// TwinCAT 3 PLC project PLC1
// ProgramVersion: 3.1.4024.0
// libraries:
//   Tc2_Standard, * (Beckhoff Automation GmbH)
//   Tc2_System, * (Beckhoff Automation GmbH)
//   Tc3_IotCommunicator, * (Beckhoff Automation GmbH)
//   Tc3_Module, * (Beckhoff Automation GmbH)
// project tree:
//   DUTs/ ST_Mqtt_Data.TcDUT
//   / PlcTask.TcTTO
//   POUs/ MAIN.TcPOU
// real-time tasks:
//   TASK PlcTask: cycle T#10ms, priority 20, ADS port 350

CONFIGURATION PLC1
    RESOURCE PLC ON TwinCAT3
        TASK PlcTask(INTERVAL := T#10ms, PRIORITY := 20);
        PROGRAM MAIN WITH PlcTask : MAIN;
    END_RESOURCE
END_CONFIGURATION

// ---- DUTs/ST_Mqtt_Data.TcDUT
TYPE ST_Mqtt_Data :
STRUCT
	{attribute 'iot.DisplayName' := 'Valve'}
	valve1 : BOOL;
	{attribute 'iot.DisplayName' := 'Pressure Transducer'}
    {attribute 'iot.ReadOnly' := 'true'}
    {attribute 'iot.Unit' := 'Celsius'}
	{attribute 'iot.MinValue' := '5'}
    {attribute 'iot.MaxValue' := '30'}
	pt1 : REAL;
END_STRUCT
END_TYPE

// ---- POUs/MAIN.TcPOU
PROGRAM MAIN
VAR
	fb_IotComm : FB_IotCommunicator := ( sHostName := 'broker.emqx.io',
										 nPort := 1883,
			 							 sMainTopic := 'cc_test',
			 							 sDeviceName := 'adrian_laptop',
			 							 sUser := 'asita',
			 							 sPassword := 'ccinc');
	mqtt_data : ST_Mqtt_Data;
	tmrSend : TON;
END_VAR

fb_IotComm.Execute(TRUE);

tmrSend(IN := NOT tmrSend.Q, PT := T#500MS);

IF fb_IotComm.bConnected AND tmrSend.Q THEN
	fb_IotComm.SendData(ADR(mqtt_data),SIZEOF(mqtt_data));
END_IF

END_PROGRAM
